FUNCTION_BLOCK FBLED
VAR_INPUT
END_VAR
VAR_OUTPUT
END_VAR
VAR
END_VAR

END_FUNCTION_BLOCK

(* stored: Version 1.1.0.1, ProductVersion 3.1.4026.18
   POU FBLED: Id {e5242f04-1ceb-4b87-b629-e1c7ae9092ab}, SpecialFunc None *)
